{attribute addProperty BoxType "EJ1914-0000-0017"}
{attribute addProperty Id "FSoE_CommandUSINT811FSIN_Module_1_ErrAckBIT10.1251FSIN_Module_2_ErrAckBIT10.1251FSoE_CRC_000UINT1623FSoE_Connection_IDUINT1622"}
{attribute addProperty CRC "669256817"}
{attribute addProperty SizeInBites "48"}
{attribute addProperty SizeInBytes "6"}
TYPE FSOE_27E40C71 :
STRUCT
	{attribute addProperty Name "FSoE_Command"}
	FSoE_Command : USINT;
	{attribute addProperty Name "FSIN_Module_1_ErrAck"}
	FSIN_Module_1_ErrAck : BOOL;
	{attribute addProperty Name "FSIN_Module_2_ErrAck"}
	FSIN_Module_2_ErrAck : BOOL;
	{attribute 'hide'}
	reserve_1_BIT_0 : BOOL;
	{attribute 'hide'}
	reserve_1_BIT_1 : BOOL;
	{attribute 'hide'}
	reserve_1_BIT_2 : BOOL;
	{attribute 'hide'}
	reserve_1_BIT_3 : BOOL;
	{attribute 'hide'}
	reserve_1_BIT_4 : BOOL;
	{attribute 'hide'}
	reserve_1_BIT_5 : BOOL;
	{attribute addProperty Name "FSoE_CRC_000"}
	FSoE_CRC_000 : UINT;
	{attribute addProperty Name "FSoE_Connection_ID"}
	FSoE_Connection_ID : UINT;
END_STRUCT
END_TYPE

(* stored: Version 1.2.0.0, ProductVersion 3.1.4024.9
   DUT FSOE_27E40C71: Id {ebac517b-dcf3-4372-b446-b641d78707e5} *)
